FUNCTION_BLOCK SERVER_3_1 (* 3 SD/1 RD Server Interface *)
  (* Standard: 61499-1; Classification: Communications *)
  (* Version 0.0, 2005-06-11, JHC, Holobloc Inc *)
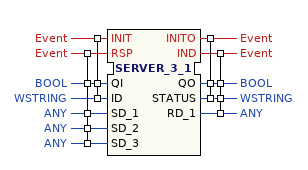
  EVENT_INPUT
    INIT WITH QI, ID;
    RSP WITH QI, SD_1, SD_2, SD_3;
  END_EVENT
  EVENT_OUTPUT
    INITO WITH QO, STATUS;
    IND WITH QO, STATUS, RD_1;
  END_EVENT
  VAR_INPUT
    QI : BOOL;
    ID : WSTRING;
    SD_1 : ANY;
    SD_2 : ANY;
    SD_3 : ANY;
  END_VAR
  VAR_OUTPUT
    QO : BOOL;
    STATUS : WSTRING;
    RD_1 : ANY;
  END_VAR
END_FUNCTION_BLOCK
